// Writes a length (in bytes) for length-delimited data.
FUNCTION F_WriteLength : HRESULT
VAR_IN_OUT CONSTANT
    aBuffer : ARRAY [*] OF BYTE;   
END_VAR
VAR_IN_OUT
    stState : ST_WriterInternalState;
END_VAR
VAR_INPUT
    nLength : UDINT;
END_VAR

{warning disable C0041}
F_WriteLength := F_WriteRawVarint32(aBuffer, stState, nLength);

END_FUNCTION

(* stored: Version 1.1.0.1
   POU F_WriteLength: Id {07f3f053-aeab-4a55-bb4b-e3a63873a37e}, SpecialFunc None *)
